///#########################################################
///Main POU for TCP/IP based EPICS-interface. The TCP/IP server related code is based on Beckhoff sample code. Changes and additions have been made to this code for the general purpose EPICS interface.
///
///	Library:		
///	
///
///	Global Variables:
///	- EPICS_MAX_FRAME_SIZE					
///	- EPICS_ARRAY_DELIMITER					
///	- EPICS_COMMAND_DELIMITER
/// - PLCPRJ_BUFFER_SIZE				 
///
///	Data types:
///	
///	External functions:
///		- TC2_Standard lib
///		- Tc2_Utilities lib
///		- Tc2_System lib
///		
///
///###########################################################

PROGRAM MAIN
VAR
	sVersion: STRING:='0.9.1';
END_VAR
VAR
	sSrvNetID	: T_AmsNetID	:= '';(* TwinCAT TCP/IP server network address *)
	bEnable		: BOOL := TRUE;(* TRUE => Enable server data exchange, FALSE => Disable *)
	bLog		: BOOL := FALSE;(* TRUE => Enable message/error log, FALSE => Disable *)
	
	fbServer	: FB_Server := ( 	sLocalHost :=  '0.0.0.0' (*Own (server) IP address!  '192.168.40.106'*), 
									nLocalPort := 5000,(* Own (server) port number! *) 
									sPrefix := 'SERVER::' );

	fbCloseAll	: FB_SocketCloseAll;
	bInitialize	: BOOL := TRUE;
	
	//Included utilities in EpicsComModule
	fbNTShutdown: NT_Shutdown;
	fbNTAbortShutdown:NT_AbortShutdown;
	iCounter:INT:=0;
END_VAR

//Delay execution
IF EPICS_SAMPLE_TIME>100 THEN
	EPICS_SAMPLE_TIME:=100;
ELSIF  EPICS_SAMPLE_TIME<1 THEN
	EPICS_SAMPLE_TIME:=1;	
END_IF

iCounter:=iCounter+1;
IF iCounter>=EPICS_SAMPLE_TIME THEN  //Possability to change communcation execution speed from EPICS (via the global variable EPICS_SAMPLE_TIME)
	iCounter:=0;
	(* On PLC reset or program download close all created/opened sockets/connections *)
	fbCloseAll( sSrvNetID := sSrvNetID, bExecute:= bInitialize );
	IF fbCloseAll.bBusy OR fbCloseAll.bError THEN
		RETURN;
	END_IF
	bInitialize := FALSE;
	fbServer( sSrvNetID := sSrvNetID, bEnable := bEnable, bLog := bLog );
END_IF

//Execution of utilities Action
Utilities();

ACTION Utilities:
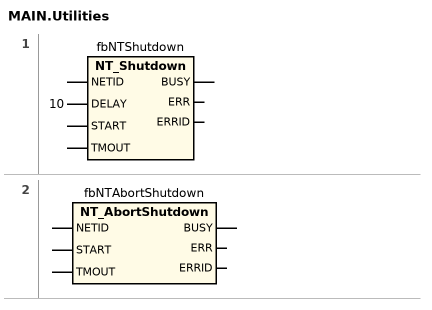
// NETWORK 1
//   fbNTShutdown: Included utilities in EpicsComModule
fbNTShutdown(DELAY := 10); // NT_Shutdown

// NETWORK 2
fbNTAbortShutdown(); // NT_AbortShutdown
END_ACTION

END_PROGRAM

(* stored: Version 1.1.0.1, ProductVersion 3.1.0.36
   POU MAIN: Id {7b6efa2b-c8d0-4c9b-b40c-faa65e5b128e}, SpecialFunc None
   Action Utilities: Id {3fe46f27-cd70-420a-b970-da286be3b9dc} *)
